FUNCTION_BLOCK FB_FlPos
VAR_INPUT
    vix_Sig : BOOL;
END_VAR
VAR_OUTPUT
    vqx_FlPos : BOOL;
END_VAR
VAR
    vsx_LastSig : BOOL;
END_VAR

vqx_FlPos := (vix_Sig = TRUE) AND (vsx_LastSig = FALSE);
vsx_LastSig := vix_Sig;

END_FUNCTION_BLOCK

(* stored: Version 1.1.0.1
   POU FB_FlPos: Id {026a26e0-becc-48e5-967e-9ba209645323}, SpecialFunc None *)
